Fanuc KAREL source: ks00038.KL

-- PROVISIONAL review KL for V1013-1; original PC SHA256 cc83a74ce60960eca049550218f61234e492aa97ecc42644cd405d6866d01645
-- Incomplete behavior may be omitted. Consult companion uncertainty JSON. Do not deploy.
PROGRAM KS00038
%NOLOCKGROUP
BEGIN
  -- UNRESOLVED_PC offsets 5-13; opcodes 3F,75
  -- UNRESOLVED_PC offsets 18-27; opcodes 3F,75
  -- UNRESOLVED_PC offsets 32-46; opcodes 22,22,1E
  -- UNRESOLVED_PC offsets 51-55; opcodes 7F
END KS00038
